SUBAPPLICATION Uebung_079 (* alle TECU FBs *)
  (* Standard: 61499-2; Description: Copyright (c) 2023 Meisterschulen am Ostbahnhof This program and the accompanying materials are made available under the terms of the Eclipse Public License 2.0 which is available at https://www.eclipse.org/legal/epl-2.0/ SPDX-License-Identifier: EPL-2.0 *)
  (* Version 1.0, 2023-10-23, Franz Höpfinger, Meisterschulen am Ostbahnhof *)
  PACKAGE Uebungen;
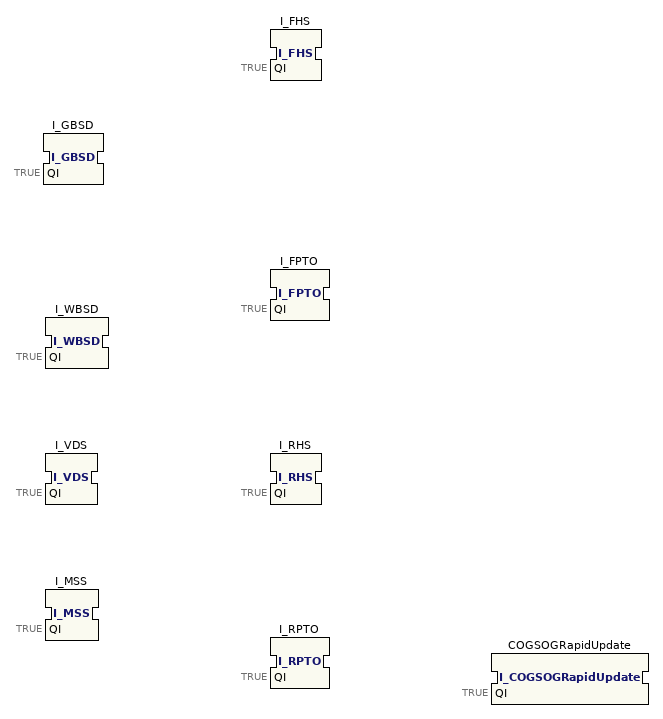
  FBS
    I_GBSD : isobus::tecu::I_GBSD(QI := TRUE);
    I_VDS : isobus::tecu::I_VDS(QI := TRUE);
    I_WBSD : isobus::tecu::I_WBSD(QI := TRUE);
    I_MSS : isobus::tecu::I_MSS(QI := TRUE);
    I_FHS : isobus::tecu::I_FHS(QI := TRUE);
    I_FPTO : isobus::tecu::I_FPTO(QI := TRUE);
    I_RHS : isobus::tecu::I_RHS(QI := TRUE);
    I_RPTO : isobus::tecu::I_RPTO(QI := TRUE);
    COGSOGRapidUpdate : isobus::tecu::I_COGSOGRapidUpdate(QI := TRUE);
  END_FBS
END_SUBAPPLICATION
